      Area03_Messages.W.Msg[WngIndex + 0] := A0301_Ribaltatore.Warning.Ax.NotAutReady;
      Area03_Messages.W.Msg[WngIndex + 1] := A0301_Ribaltatore.Warning.Ax.Minus_CndMissing;
      Area03_Messages.W.Msg[WngIndex + 2] := A0301_Ribaltatore.Warning.Ax.Plus_CndMissing AND A0301_Ribaltatore.COut.Solleva_Rib.Work;
      Area03_Messages.W.Msg[WngIndex + 3] := A0301_Ribaltatore.Warning.Ax.S120_Warning;
      Area03_Messages.W.Msg[WngIndex + 4] := A0301_Ribaltatore.Warning.Ax.Ax_NotHomed;
      Area03_Messages.W.Msg[WngIndex + 5] := A0301_Ribaltatore.Warning.Ax.Ax_FlyingHome;
      Area03_Messages.W.Msg[WngIndex + 6] := A0301_Ribaltatore.Warning.Ax.Ax_SwLimitMinus;
      Area03_Messages.W.Msg[WngIndex + 7] := A0301_Ribaltatore.Warning.Ax.Ax_SwLimitPlus;
      Area03_Messages.W.Msg[WngIndex + 8] := A0301_Ribaltatore.Warning.OP_REST_MissingCnd;
      Area03_Messages.W.Msg[WngIndex + 9] := A0301_Ribaltatore.Warning.OP_WORK_MissingCnd;
      Area03_Messages.W.Msg[WngIndex + 10] := A0301_Ribaltatore.Warning.Solleva_Rib[1].NotAutReady;
      Area03_Messages.W.Msg[WngIndex + 11] := A0301_Ribaltatore.Warning.Solleva_Rib[1].PressureRunning_Timeout;
      Area03_Messages.W.Msg[WngIndex + 12] := A0301_Ribaltatore.Warning.Solleva_Rib[1].Rest_MissingExtEnable;
      Area03_Messages.W.Msg[WngIndex + 13] := A0301_Ribaltatore.Warning.Solleva_Rib[1].Work_MissingExtEnable;
      Area03_Messages.W.Msg[WngIndex + 14] := A0301_Ribaltatore.Warning.Solleva_Rib[1].Missing_Rest_Ls_ON[1];
      Area03_Messages.W.Msg[WngIndex + 15] := A0301_Ribaltatore.Warning.Solleva_Rib[1].Missing_Work_Ls_ON[1];
      Area03_Messages.W.Msg[WngIndex + 16] := A0301_Ribaltatore.Warning.Solleva_Rib[2].NotAutReady;
      Area03_Messages.W.Msg[WngIndex + 17] := A0301_Ribaltatore.Warning.Solleva_Rib[2].PressureRunning_Timeout;
      Area03_Messages.W.Msg[WngIndex + 18] := A0301_Ribaltatore.Warning.Solleva_Rib[2].Rest_MissingExtEnable;
      Area03_Messages.W.Msg[WngIndex + 19] := A0301_Ribaltatore.Warning.Solleva_Rib[2].Work_MissingExtEnable;
      Area03_Messages.W.Msg[WngIndex + 20] := A0301_Ribaltatore.Warning.Solleva_Rib[2].Missing_Rest_Ls_ON[1];
      Area03_Messages.W.Msg[WngIndex + 21] := A0301_Ribaltatore.Warning.Solleva_Rib[2].Missing_Work_Ls_ON[1];
      Area03_Messages.W.Msg[WngIndex + 22] := A0301_Ribaltatore.Warning.Solleva_Rib[3].NotAutReady;
      Area03_Messages.W.Msg[WngIndex + 23] := A0301_Ribaltatore.Warning.Solleva_Rib[3].PressureRunning_Timeout;
      Area03_Messages.W.Msg[WngIndex + 24] := A0301_Ribaltatore.Warning.Solleva_Rib[3].Rest_MissingExtEnable;
      Area03_Messages.W.Msg[WngIndex + 25] := A0301_Ribaltatore.Warning.Solleva_Rib[3].Work_MissingExtEnable;
      Area03_Messages.W.Msg[WngIndex + 26] := A0301_Ribaltatore.Warning.Solleva_Rib[3].Missing_Rest_Ls_ON[1];
      Area03_Messages.W.Msg[WngIndex + 27] := A0301_Ribaltatore.Warning.Solleva_Rib[3].Missing_Work_Ls_ON[1];
      Area03_Messages.W.Msg[WngIndex + 28] := A0301_Ribaltatore.Warning.Solleva_Rib[4].NotAutReady;
      Area03_Messages.W.Msg[WngIndex + 29] := A0301_Ribaltatore.Warning.Solleva_Rib[4].PressureRunning_Timeout;
      Area03_Messages.W.Msg[WngIndex + 30] := A0301_Ribaltatore.Warning.Solleva_Rib[4].Rest_MissingExtEnable;
      Area03_Messages.W.Msg[WngIndex + 31] := A0301_Ribaltatore.Warning.Solleva_Rib[4].Work_MissingExtEnable;
      Area03_Messages.W.Msg[WngIndex + 32] := A0301_Ribaltatore.Warning.Solleva_Rib[4].Missing_Rest_Ls_ON[1];
      Area03_Messages.W.Msg[WngIndex + 33] := A0301_Ribaltatore.Warning.Solleva_Rib[4].Missing_Work_Ls_ON[1];
      Area03_Messages.W.Msg[WngIndex + 34] := A0301_Ribaltatore.Warning.Solleva_Rib[5].NotAutReady;
      Area03_Messages.W.Msg[WngIndex + 35] := A0301_Ribaltatore.Warning.Solleva_Rib[5].PressureRunning_Timeout;
      Area03_Messages.W.Msg[WngIndex + 36] := A0301_Ribaltatore.Warning.Solleva_Rib[5].Rest_MissingExtEnable;
      Area03_Messages.W.Msg[WngIndex + 37] := A0301_Ribaltatore.Warning.Solleva_Rib[5].Work_MissingExtEnable;
      Area03_Messages.W.Msg[WngIndex + 38] := A0301_Ribaltatore.Warning.Solleva_Rib[5].Missing_Rest_Ls_ON[1];
      Area03_Messages.W.Msg[WngIndex + 39] := A0301_Ribaltatore.Warning.Solleva_Rib[5].Missing_Work_Ls_ON[1];
      Area03_Messages.W.Msg[WngIndex + 40] := A0301_Ribaltatore.Warning.Solleva_Rib[6].NotAutReady;
      Area03_Messages.W.Msg[WngIndex + 41] := A0301_Ribaltatore.Warning.Solleva_Rib[6].PressureRunning_Timeout;
      Area03_Messages.W.Msg[WngIndex + 42] := A0301_Ribaltatore.Warning.Solleva_Rib[6].Rest_MissingExtEnable;
      Area03_Messages.W.Msg[WngIndex + 43] := A0301_Ribaltatore.Warning.Solleva_Rib[6].Work_MissingExtEnable;
      Area03_Messages.W.Msg[WngIndex + 44] := A0301_Ribaltatore.Warning.Solleva_Rib[6].Missing_Rest_Ls_ON[1];
      Area03_Messages.W.Msg[WngIndex + 45] := A0301_Ribaltatore.Warning.Solleva_Rib[6].Missing_Work_Ls_ON[1];
      Area03_Messages.W.Msg[WngIndex + 46] := FALSE;
      Area03_Messages.W.Msg[WngIndex + 47] := FALSE;
      Area03_Messages.W.Msg[WngIndex + 48] := FALSE;
      Area03_Messages.W.Msg[WngIndex + 49] := FALSE;

      //Fermi P4
      //
      WngIndex := 280;

      Area03_Messages.W.Msg[WngIndex + 0] := A0301_Fermi_P4.Warning.Fermi[1].NotAutReady;
      Area03_Messages.W.Msg[WngIndex + 1] := A0301_Fermi_P4.Warning.Fermi[1].PressureRunning_Timeout;
      Area03_Messages.W.Msg[WngIndex + 2] := A0301_Fermi_P4.Warning.Fermi[1].Rest_MissingExtEnable;
      Area03_Messages.W.Msg[WngIndex + 3] := A0301_Fermi_P4.Warning.Fermi[1].Work_MissingExtEnable;
      Area03_Messages.W.Msg[WngIndex + 4] := A0301_Fermi_P4.Warning.Fermi[1].Missing_Rest_Ls_ON[1];
      Area03_Messages.W.Msg[WngIndex + 5] := A0301_Fermi_P4.Warning.Fermi[1].Missing_Work_Ls_ON[1];
      Area03_Messages.W.Msg[WngIndex + 6] := A0301_Fermi_P4.Warning.Fermi[2].NotAutReady;
      Area03_Messages.W.Msg[WngIndex + 7] := A0301_Fermi_P4.Warning.Fermi[2].PressureRunning_Timeout;
      Area03_Messages.W.Msg[WngIndex + 8] := A0301_Fermi_P4.Warning.Fermi[2].Rest_MissingExtEnable;
      Area03_Messages.W.Msg[WngIndex + 9] := A0301_Fermi_P4.Warning.Fermi[2].Work_MissingExtEnable;
      Area03_Messages.W.Msg[WngIndex + 10] := A0301_Fermi_P4.Warning.Fermi[2].Missing_Rest_Ls_ON[1];
      Area03_Messages.W.Msg[WngIndex + 11] := A0301_Fermi_P4.Warning.Fermi[2].Missing_Work_Ls_ON[1];
      Area03_Messages.W.Msg[WngIndex + 12] := A0301_Fermi_P4.Warning.Fermi[3].NotAutReady;
      Area03_Messages.W.Msg[WngIndex + 13] := A0301_Fermi_P4.Warning.Fermi[3].PressureRunning_Timeout;
      Area03_Messages.W.Msg[WngIndex + 14] := A0301_Fermi_P4.Warning.Fermi[3].Rest_MissingExtEnable;
      Area03_Messages.W.Msg[WngIndex + 15] := A0301_Fermi_P4.Warning.Fermi[3].Work_MissingExtEnable;
      Area03_Messages.W.Msg[WngIndex + 16] := A0301_Fermi_P4.Warning.Fermi[3].Missing_Rest_Ls_ON[1];
      Area03_Messages.W.Msg[WngIndex + 17] := A0301_Fermi_P4.Warning.Fermi[3].Missing_Work_Ls_ON[1];
      Area03_Messages.W.Msg[WngIndex + 18] := A0301_Fermi_P4.Warning.Fermi[4].NotAutReady;
      Area03_Messages.W.Msg[WngIndex + 19] := A0301_Fermi_P4.Warning.Fermi[4].PressureRunning_Timeout;
      Area03_Messages.W.Msg[WngIndex + 20] := A0301_Fermi_P4.Warning.Fermi[4].Rest_MissingExtEnable;
      Area03_Messages.W.Msg[WngIndex + 21] := A0301_Fermi_P4.Warning.Fermi[4].Work_MissingExtEnable;
      Area03_Messages.W.Msg[WngIndex + 22] := A0301_Fermi_P4.Warning.Fermi[4].Missing_Rest_Ls_ON[1];
      Area03_Messages.W.Msg[WngIndex + 23] := A0301_Fermi_P4.Warning.Fermi[4].Missing_Work_Ls_ON[1];
      Area03_Messages.W.Msg[WngIndex + 24] := A0301_Fermi_P4.Warning.Fermi[5].NotAutReady;
      Area03_Messages.W.Msg[WngIndex + 25] := A0301_Fermi_P4.Warning.Fermi[5].PressureRunning_Timeout;
      Area03_Messages.W.Msg[WngIndex + 26] := A0301_Fermi_P4.Warning.Fermi[5].Rest_MissingExtEnable;
      Area03_Messages.W.Msg[WngIndex + 27] := A0301_Fermi_P4.Warning.Fermi[5].Work_MissingExtEnable;
      Area03_Messages.W.Msg[WngIndex + 28] := A0301_Fermi_P4.Warning.Fermi[5].Missing_Rest_Ls_ON[1];
      Area03_Messages.W.Msg[WngIndex + 29] := A0301_Fermi_P4.Warning.Fermi[5].Missing_Work_Ls_ON[1];
      Area03_Messages.W.Msg[WngIndex + 30] := A0301_Fermi_P4.Warning.Fermi[6].NotAutReady;
      Area03_Messages.W.Msg[WngIndex + 31] := A0301_Fermi_P4.Warning.Fermi[6].PressureRunning_Timeout;
      Area03_Messages.W.Msg[WngIndex + 32] := A0301_Fermi_P4.Warning.Fermi[6].Rest_MissingExtEnable;
      Area03_Messages.W.Msg[WngIndex + 33] := A0301_Fermi_P4.Warning.Fermi[6].Work_MissingExtEnable;
      Area03_Messages.W.Msg[WngIndex + 34] := A0301_Fermi_P4.Warning.Fermi[6].Missing_Rest_Ls_ON[1];
      Area03_Messages.W.Msg[WngIndex + 35] := A0301_Fermi_P4.Warning.Fermi[6].Missing_Work_Ls_ON[1];
      Area03_Messages.W.Msg[WngIndex + 36] := FALSE;
      Area03_Messages.W.Msg[WngIndex + 37] := FALSE;
      Area03_Messages.W.Msg[WngIndex + 38] := A0301_Fermi_P4.Warning.OP_REST_MissingCnd;
      Area03_Messages.W.Msg[WngIndex + 39] := A0301_Fermi_P4.Warning.OP_WORK_MissingCnd;

      //Spintore Laterale
      //
      WngIndex := 330;

      Area03_Messages.W.Msg[WngIndex + 0] := A0301_Spintore_Lat.Warning.Vrt_1.NotAutReady;
      Area03_Messages.W.Msg[WngIndex + 1] := A0301_Spintore_Lat.Warning.Vrt_1.PressureRunning_Timeout;
      Area03_Messages.W.Msg[WngIndex + 2] := A0301_Spintore_Lat.Warning.Vrt_1.Rest_MissingExtEnable;
      Area03_Messages.W.Msg[WngIndex + 3] := A0301_Spintore_Lat.Warning.Vrt_1.Work_MissingExtEnable;
      Area03_Messages.W.Msg[WngIndex + 4] := A0301_Spintore_Lat.Warning.Vrt_1.Missing_Rest_Ls_ON[1];
      Area03_Messages.W.Msg[WngIndex + 5] := A0301_Spintore_Lat.Warning.Vrt_1.Missing_Work_Ls_ON[1];
      Area03_Messages.W.Msg[WngIndex + 6] := FALSE;
      Area03_Messages.W.Msg[WngIndex + 7] := A0301_Spintore_Lat.Warning.Orz_1.NotAutReady;;
      Area03_Messages.W.Msg[WngIndex + 8] := A0301_Spintore_Lat.Warning.Orz_1.PressureRunning_Timeout;
      Area03_Messages.W.Msg[WngIndex + 9] := A0301_Spintore_Lat.Warning.Orz_1.Rest_MissingExtEnable;
      Area03_Messages.W.Msg[WngIndex + 10] := A0301_Spintore_Lat.Warning.Orz_1.Work_MissingExtEnable;
      Area03_Messages.W.Msg[WngIndex + 11] := A0301_Spintore_Lat.Warning.Orz_1.Missing_Rest_Ls_ON[1];
      Area03_Messages.W.Msg[WngIndex + 12] := A0301_Spintore_Lat.Warning.Orz_1.Missing_Work_Ls_ON[1];
      Area03_Messages.W.Msg[WngIndex + 13] := FALSE;
      Area03_Messages.W.Msg[WngIndex + 14] := A0301_Spintore_Lat.Warning.Orz_1_AnalSens.SensorDisabled;
      Area03_Messages.W.Msg[WngIndex + 15] := A0301_Spintore_Lat.Warning.Orz_1_AnalSens.PresetNeed;;
      Area03_Messages.W.Msg[WngIndex + 16] := A0301_Spintore_Lat.Warning.Orz_1_AnalSens.SignalError;
      Area03_Messages.W.Msg[WngIndex + 17] := FALSE;
      Area03_Messages.W.Msg[WngIndex + 18] := A0301_Spintore_Lat.Warning.OP_REST_MissingCnd;
      Area03_Messages.W.Msg[WngIndex + 19] := A0301_Spintore_Lat.Warning.OP_WORK_MissingCnd;
      Area03_Messages.W.Msg[WngIndex + 20] := A0301_Spintore_Lat.Warning.Vrt_2.NotAutReady;;
      Area03_Messages.W.Msg[WngIndex + 21] := A0301_Spintore_Lat.Warning.Vrt_2.PressureRunning_Timeout;
      Area03_Messages.W.Msg[WngIndex + 22] := A0301_Spintore_Lat.Warning.Vrt_2.Rest_MissingExtEnable;
      Area03_Messages.W.Msg[WngIndex + 23] := A0301_Spintore_Lat.Warning.Vrt_2.Work_MissingExtEnable;
      Area03_Messages.W.Msg[WngIndex + 24] := A0301_Spintore_Lat.Warning.Vrt_2.Missing_Rest_Ls_ON[1];
      Area03_Messages.W.Msg[WngIndex + 25] := A0301_Spintore_Lat.Warning.Vrt_2.Missing_Work_Ls_ON[1];
      Area03_Messages.W.Msg[WngIndex + 26] := FALSE;
      Area03_Messages.W.Msg[WngIndex + 27] := A0301_Spintore_Lat.Warning.Orz_2.NotAutReady;
      Area03_Messages.W.Msg[WngIndex + 28] := A0301_Spintore_Lat.Warning.Orz_2.PressureRunning_Timeout;
      Area03_Messages.W.Msg[WngIndex + 29] := A0301_Spintore_Lat.Warning.Orz_2.Rest_MissingExtEnable;
      Area03_Messages.W.Msg[WngIndex + 30] := A0301_Spintore_Lat.Warning.Orz_2.Work_MissingExtEnable;
      Area03_Messages.W.Msg[WngIndex + 31] := A0301_Spintore_Lat.Warning.Orz_2.Missing_Rest_Ls_ON[1];
      Area03_Messages.W.Msg[WngIndex + 32] := A0301_Spintore_Lat.Warning.Orz_2.Missing_Work_Ls_ON[1];
      Area03_Messages.W.Msg[WngIndex + 33] := A0301_Spintore_Lat.Warning.Orz_2_AnalSens.SensorDisabled;
      Area03_Messages.W.Msg[WngIndex + 34] := A0301_Spintore_Lat.Warning.Orz_2_AnalSens.PresetNeed;
      Area03_Messages.W.Msg[WngIndex + 35] := A0301_Spintore_Lat.Warning.Orz_2_AnalSens.SignalError;
      Area03_Messages.W.Msg[WngIndex + 36] := A0301_Spintore_Lat.Warning.Finestre.SpinLat1_SpinLong_Stop;
      Area03_Messages.W.Msg[WngIndex + 37] := A0301_Spintore_Lat.Warning.Finestre.SpinLat2_SpinLong_Stop;


      //Spintore Longitudinale
      //
      WngIndex := 380;

      Area03_Messages.W.Msg[WngIndex + 0] := A0301_Spintore_Lat.Warning.Sollevatori[1].NotAutReady;
      Area03_Messages.W.Msg[WngIndex + 1] := A0301_Spintore_Lat.Warning.Sollevatori[1].PressureRunning_Timeout;
      Area03_Messages.W.Msg[WngIndex + 2] := A0301_Spintore_Lat.Warning.Sollevatori[1].Rest_MissingExtEnable;
      Area03_Messages.W.Msg[WngIndex + 3] := A0301_Spintore_Lat.Warning.Sollevatori[1].Work_MissingExtEnable;
      Area03_Messages.W.Msg[WngIndex + 4] := A0301_Spintore_Lat.Warning.Sollevatori[1].Missing_Rest_Ls_ON[1];
      Area03_Messages.W.Msg[WngIndex + 5] := A0301_Spintore_Lat.Warning.Sollevatori[1].Missing_Work_Ls_ON[1];
      Area03_Messages.W.Msg[WngIndex + 6] := FALSE;
      Area03_Messages.W.Msg[WngIndex + 7] := A0301_Spintore_Lat.Warning.Sollevatori[2].NotAutReady;;
      Area03_Messages.W.Msg[WngIndex + 8] := A0301_Spintore_Lat.Warning.Sollevatori[2].PressureRunning_Timeout;
      Area03_Messages.W.Msg[WngIndex + 9] := A0301_Spintore_Lat.Warning.Sollevatori[2].Rest_MissingExtEnable;
      Area03_Messages.W.Msg[WngIndex + 10] := A0301_Spintore_Lat.Warning.Sollevatori[2].Work_MissingExtEnable;
      Area03_Messages.W.Msg[WngIndex + 11] := A0301_Spintore_Lat.Warning.Sollevatori[2].Missing_Rest_Ls_ON[1];
      Area03_Messages.W.Msg[WngIndex + 12] := A0301_Spintore_Lat.Warning.Sollevatori[2].Missing_Work_Ls_ON[1];
      Area03_Messages.W.Msg[WngIndex + 13] := FALSE;
      Area03_Messages.W.Msg[WngIndex + 14] := A0301_Spintore_Lat.Warning.Sollevatori[3].NotAutReady;
      Area03_Messages.W.Msg[WngIndex + 15] := A0301_Spintore_Lat.Warning.Sollevatori[3].PressureRunning_Timeout;
      Area03_Messages.W.Msg[WngIndex + 16] := A0301_Spintore_Lat.Warning.Sollevatori[3].Rest_MissingExtEnable;
      Area03_Messages.W.Msg[WngIndex + 17] := A0301_Spintore_Lat.Warning.Sollevatori[3].Work_MissingExtEnable;
      Area03_Messages.W.Msg[WngIndex + 18] := A0301_Spintore_Lat.Warning.Sollevatori[3].Missing_Rest_Ls_ON[1];
      Area03_Messages.W.Msg[WngIndex + 19] := A0301_Spintore_Lat.Warning.Sollevatori[3].Missing_Work_Ls_ON[1];
      Area03_Messages.W.Msg[WngIndex + 20] := FALSE;
      Area03_Messages.W.Msg[WngIndex + 21] := A0301_Spintore_Lat.Warning.Sollevatori[4].NotAutReady;
      Area03_Messages.W.Msg[WngIndex + 22] := A0301_Spintore_Lat.Warning.Sollevatori[4].PressureRunning_Timeout;
      Area03_Messages.W.Msg[WngIndex + 23] := A0301_Spintore_Lat.Warning.Sollevatori[4].Rest_MissingExtEnable;
      Area03_Messages.W.Msg[WngIndex + 24] := A0301_Spintore_Lat.Warning.Sollevatori[4].Work_MissingExtEnable;
      Area03_Messages.W.Msg[WngIndex + 25] := A0301_Spintore_Lat.Warning.Sollevatori[4].Missing_Rest_Ls_ON[1];
      Area03_Messages.W.Msg[WngIndex + 26] := A0301_Spintore_Lat.Warning.Sollevatori[4].Missing_Work_Ls_ON[1];
      Area03_Messages.W.Msg[WngIndex + 27] := FALSE;
      Area03_Messages.W.Msg[WngIndex + 28] := A0301_Spintore_Lat.Warning.Sollevatori[5].NotAutReady;
      Area03_Messages.W.Msg[WngIndex + 29] := A0301_Spintore_Lat.Warning.Sollevatori[5].PressureRunning_Timeout;
      Area03_Messages.W.Msg[WngIndex + 30] := A0301_Spintore_Lat.Warning.Sollevatori[5].Rest_MissingExtEnable;
      Area03_Messages.W.Msg[WngIndex + 31] := A0301_Spintore_Lat.Warning.Sollevatori[5].Work_MissingExtEnable;
      Area03_Messages.W.Msg[WngIndex + 32] := A0301_Spintore_Lat.Warning.Sollevatori[5].Missing_Rest_Ls_ON[1];
      Area03_Messages.W.Msg[WngIndex + 33] := A0301_Spintore_Lat.Warning.Sollevatori[5].Missing_Work_Ls_ON[1];
      Area03_Messages.W.Msg[WngIndex + 34] := FALSE;
      Area03_Messages.W.Msg[WngIndex + 35] := A0301_Spintore_Lat.Warning.Sollevatori[6].NotAutReady;
      Area03_Messages.W.Msg[WngIndex + 36] := A0301_Spintore_Lat.Warning.Sollevatori[6].PressureRunning_Timeout;
      Area03_Messages.W.Msg[WngIndex + 37] := A0301_Spintore_Lat.Warning.Sollevatori[6].Rest_MissingExtEnable;
      Area03_Messages.W.Msg[WngIndex + 38] := A0301_Spintore_Lat.Warning.Sollevatori[6].Work_MissingExtEnable;
      Area03_Messages.W.Msg[WngIndex + 39] := A0301_Spintore_Lat.Warning.Sollevatori[6].Missing_Rest_Ls_ON[1];
      Area03_Messages.W.Msg[WngIndex + 40] := A0301_Spintore_Lat.Warning.Sollevatori[6].Missing_Work_Ls_ON[1];
      Area03_Messages.W.Msg[WngIndex + 41] := FALSE;
      Area03_Messages.W.Msg[WngIndex + 42] := A0301_Spintore_Lat.Warning.Sollevatori[7].NotAutReady;
      Area03_Messages.W.Msg[WngIndex + 43] := A0301_Spintore_Lat.Warning.Sollevatori[7].PressureRunning_Timeout;
      Area03_Messages.W.Msg[WngIndex + 44] := A0301_Spintore_Lat.Warning.Sollevatori[7].Rest_MissingExtEnable;
      Area03_Messages.W.Msg[WngIndex + 45] := A0301_Spintore_Lat.Warning.Sollevatori[7].Work_MissingExtEnable;
      Area03_Messages.W.Msg[WngIndex + 46] := A0301_Spintore_Lat.Warning.Sollevatori[7].Missing_Rest_Ls_ON[1];
      Area03_Messages.W.Msg[WngIndex + 47] := A0301_Spintore_Lat.Warning.Sollevatori[7].Missing_Work_Ls_ON[1];
      Area03_Messages.W.Msg[WngIndex + 48] := FALSE;
      Area03_Messages.W.Msg[WngIndex + 49] := FALSE;



      //Manager stazioni pareggiamento
      //
      WngIndex := 430;

      Area03_Messages.W.Msg[WngIndex + 0] := A0302_Manager.Warning.CheckBancoAccumulo;
      Area03_Messages.W.Msg[WngIndex + 1] := FALSE;
      Area03_Messages.W.Msg[WngIndex + 2] := FALSE;
      Area03_Messages.W.Msg[WngIndex + 3] := FALSE;
      Area03_Messages.W.Msg[WngIndex + 4] := FALSE;
      Area03_Messages.W.Msg[WngIndex + 5] := FALSE;
      Area03_Messages.W.Msg[WngIndex + 6] := FALSE;
      Area03_Messages.W.Msg[WngIndex + 7] := FALSE;
      Area03_Messages.W.Msg[WngIndex + 8] := FALSE;
      Area03_Messages.W.Msg[WngIndex + 9] := FALSE;

      //HU CYTROPACK
      //
      WngIndex := 440;

      Area03_Messages.W.Msg[WngIndex + 0] := FALSE;
      Area03_Messages.W.Msg[WngIndex + 1] := FALSE;
      Area03_Messages.W.Msg[WngIndex + 2] := FALSE;
      Area03_Messages.W.Msg[WngIndex + 3] := FALSE;
      Area03_Messages.W.Msg[WngIndex + 4] := FALSE;
      Area03_Messages.W.Msg[WngIndex + 5] := FALSE;
      Area03_Messages.W.Msg[WngIndex + 6] := FALSE;
      Area03_Messages.W.Msg[WngIndex + 7] := FALSE;
      Area03_Messages.W.Msg[WngIndex + 8] := FALSE;
      Area03_Messages.W.Msg[WngIndex + 9] := FALSE;
      Area03_Messages.W.Msg[WngIndex + 10] := FALSE;
      Area03_Messages.W.Msg[WngIndex + 11] := FALSE;
      Area03_Messages.W.Msg[WngIndex + 12] := FALSE;
      Area03_Messages.W.Msg[WngIndex + 13] := FALSE;
      Area03_Messages.W.Msg[WngIndex + 14] := FALSE;
      Area03_Messages.W.Msg[WngIndex + 15] := FALSE;
      Area03_Messages.W.Msg[WngIndex + 16] := FALSE;
      Area03_Messages.W.Msg[WngIndex + 17] := FALSE;
      Area03_Messages.W.Msg[WngIndex + 18] := FALSE;
      Area03_Messages.W.Msg[WngIndex + 19] := FALSE;

      //Spintore
      //
      WngIndex := 470;

      Area03_Messages.W.Msg[WngIndex + 0] := A0302_Spintore.Warning.Ax.NotAutReady;
      Area03_Messages.W.Msg[WngIndex + 1] := A0302_Spintore.Warning.Ax.Minus_CndMissing;
      Area03_Messages.W.Msg[WngIndex + 2] := A0302_Spintore.Warning.Ax.Plus_CndMissing;
      Area03_Messages.W.Msg[WngIndex + 3] := A0302_Spintore.Warning.Ax.S120_Warning;
      Area03_Messages.W.Msg[WngIndex + 4] := A0302_Spintore.Warning.Ax.Ax_NotHomed;
      Area03_Messages.W.Msg[WngIndex + 5] := A0302_Spintore.Warning.Ax.Ax_FlyingHome;
      Area03_Messages.W.Msg[WngIndex + 6] := A0302_Spintore.Warning.Ax.Ax_SwLimitMinus;
      Area03_Messages.W.Msg[WngIndex + 7] := A0302_Spintore.Warning.Ax.Ax_SwLimitPlus;
      Area03_Messages.W.Msg[WngIndex + 8] := FALSE;
      Area03_Messages.W.Msg[WngIndex + 9] := FALSE;
      Area03_Messages.W.Msg[WngIndex + 10] := A0302_Spintore.Warning.Vrt.NotAutReady;
      Area03_Messages.W.Msg[WngIndex + 11] := A0302_Spintore.Warning.Vrt.PressureRunning_Timeout;
      Area03_Messages.W.Msg[WngIndex + 12] := A0302_Spintore.Warning.Vrt.Rest_MissingExtEnable;
      Area03_Messages.W.Msg[WngIndex + 13] := A0302_Spintore.Warning.Vrt.Work_MissingExtEnable;
      Area03_Messages.W.Msg[WngIndex + 14] := A0302_Spintore.Warning.Vrt.Missing_Rest_Ls_ON[1];
      Area03_Messages.W.Msg[WngIndex + 15] := A0302_Spintore.Warning.Vrt.Missing_Work_Ls_ON[1];
      Area03_Messages.W.Msg[WngIndex + 16] := FALSE;
      Area03_Messages.W.Msg[WngIndex + 17] := FALSE;
      Area03_Messages.W.Msg[WngIndex + 18] := A0302_Spintore.Warning.Orz.NotAutReady;
      Area03_Messages.W.Msg[WngIndex + 19] := A0302_Spintore.Warning.Orz.PressureRunning_Timeout;
      Area03_Messages.W.Msg[WngIndex + 20] := A0302_Spintore.Warning.Orz.Rest_MissingExtEnable;
      Area03_Messages.W.Msg[WngIndex + 21] := A0302_Spintore.Warning.Orz.Work_MissingExtEnable;
      Area03_Messages.W.Msg[WngIndex + 22] := A0302_Spintore.Warning.Orz.Missing_Rest_Ls_ON[1];
      Area03_Messages.W.Msg[WngIndex + 23] := A0302_Spintore.Warning.Orz.Missing_Work_Ls_ON[1];
      Area03_Messages.W.Msg[WngIndex + 24] := FALSE;
      Area03_Messages.W.Msg[WngIndex + 25] := FALSE;
      Area03_Messages.W.Msg[WngIndex + 26] := A0302_Spintore.Warning.Orz_AnalSens.SensorDisabled;
      Area03_Messages.W.Msg[WngIndex + 27] := A0302_Spintore.Warning.Orz_AnalSens.PresetNeed;
      Area03_Messages.W.Msg[WngIndex + 28] := A0302_Spintore.Warning.Orz_AnalSens.SignalError;
      Area03_Messages.W.Msg[WngIndex + 29] := FALSE;
      Area03_Messages.W.Msg[WngIndex + 30] := FALSE;
      Area03_Messages.W.Msg[WngIndex + 31] := A0302_Spintore.Warning.OP_REST_MissingCnd;
      Area03_Messages.W.Msg[WngIndex + 32] := A0302_Spintore.Warning.OP_WORK_MissingCnd;

      //Bordatrice
      //
      WngIndex := 510;

      Area03_Messages.W.Msg[WngIndex + 0] := A0302_Bordatrice.Warning.Ax.NotAutReady;
      Area03_Messages.W.Msg[WngIndex + 1] := A0302_Bordatrice.Warning.Ax.Minus_CndMissing;
      Area03_Messages.W.Msg[WngIndex + 2] := A0302_Bordatrice.Warning.Ax.Plus_CndMissing;
      Area03_Messages.W.Msg[WngIndex + 3] := A0302_Bordatrice.Warning.Ax.S120_Warning;
      Area03_Messages.W.Msg[WngIndex + 4] := A0302_Bordatrice.Warning.Ax.Ax_NotHomed;
      Area03_Messages.W.Msg[WngIndex + 5] := A0302_Bordatrice.Warning.Ax.Ax_FlyingHome;
      Area03_Messages.W.Msg[WngIndex + 6] := A0302_Bordatrice.Warning.Ax.Ax_SwLimitMinus;
      Area03_Messages.W.Msg[WngIndex + 7] := A0302_Bordatrice.Warning.Ax.Ax_SwLimitPlus;
      Area03_Messages.W.Msg[WngIndex + 8] := A0302_Bordatrice.Warning.OP_REST_MissingCnd;
      Area03_Messages.W.Msg[WngIndex + 9] := A0302_Bordatrice.Warning.OP_WORK_MissingCnd;
      Area03_Messages.W.Msg[WngIndex + 10] := FALSE;
      Area03_Messages.W.Msg[WngIndex + 11] := FALSE;
      Area03_Messages.W.Msg[WngIndex + 12] := FALSE;
      Area03_Messages.W.Msg[WngIndex + 13] := FALSE;
      Area03_Messages.W.Msg[WngIndex + 14] := FALSE;
      Area03_Messages.W.Msg[WngIndex + 15] := FALSE;
      Area03_Messages.W.Msg[WngIndex + 16] := FALSE;
      Area03_Messages.W.Msg[WngIndex + 17] := FALSE;
      Area03_Messages.W.Msg[WngIndex + 18] := FALSE;
      Area03_Messages.W.Msg[WngIndex + 19] := FALSE;
      Area03_Messages.W.Msg[WngIndex + 20] := FALSE;


      //Rulliera
      //
      WngIndex := 540;

      Area03_Messages.W.Msg[WngIndex + 0] := A0302_Rulliera.Warning.Rulliera[1].NotAutReady;
      Area03_Messages.W.Msg[WngIndex + 1] := A0302_Rulliera.Warning.Rulliera[1].MissingCnd_Bkw;
      Area03_Messages.W.Msg[WngIndex + 2] := A0302_Rulliera.Warning.Rulliera[1].MissingCnd_Fwd;
      Area03_Messages.W.Msg[WngIndex + 3] := A0302_Rulliera.Warning.Rulliera[1].Ax.Drive;
      Area03_Messages.W.Msg[WngIndex + 4] := A0302_Rulliera.Warning.Rulliera[2].NotAutReady;
      Area03_Messages.W.Msg[WngIndex + 5] := A0302_Rulliera.Warning.Rulliera[2].MissingCnd_Bkw;
      Area03_Messages.W.Msg[WngIndex + 6] := A0302_Rulliera.Warning.Rulliera[2].MissingCnd_Fwd;
      Area03_Messages.W.Msg[WngIndex + 7] := A0302_Rulliera.Warning.Rulliera[2].Ax.Drive;
      Area03_Messages.W.Msg[WngIndex + 8] := A0302_Rulliera.Warning.OP_REST_MissingCnd;
      Area03_Messages.W.Msg[WngIndex + 9] := A0302_Rulliera.Warning.OP_WORK_MissingCnd;
      Area03_Messages.W.Msg[WngIndex + 10] := FALSE;
      Area03_Messages.W.Msg[WngIndex + 11] := FALSE;
      Area03_Messages.W.Msg[WngIndex + 12] := FALSE;
      Area03_Messages.W.Msg[WngIndex + 13] := FALSE;
      Area03_Messages.W.Msg[WngIndex + 14] := FALSE;
      Area03_Messages.W.Msg[WngIndex + 15] := FALSE;
      Area03_Messages.W.Msg[WngIndex + 16] := FALSE;
      Area03_Messages.W.Msg[WngIndex + 17] := FALSE;
      Area03_Messages.W.Msg[WngIndex + 18] := FALSE;
      Area03_Messages.W.Msg[WngIndex + 19] := FALSE;


      //Centratori
      //
      WngIndex := 560;

      Area03_Messages.W.Msg[WngIndex + 0] := A0302_Centratori.Warning.Centratore[1].NotAutReady;
      Area03_Messages.W.Msg[WngIndex + 1] := A0302_Centratori.Warning.Centratore[1].PressureRunning_Timeout;
      Area03_Messages.W.Msg[WngIndex + 2] := A0302_Centratori.Warning.Centratore[1].Rest_MissingExtEnable;
      Area03_Messages.W.Msg[WngIndex + 3] := A0302_Centratori.Warning.Centratore[1].Work_MissingExtEnable;
      Area03_Messages.W.Msg[WngIndex + 4] := A0302_Centratori.Warning.Centratore[1].Missing_Rest_Ls_ON[1];
      Area03_Messages.W.Msg[WngIndex + 5] := A0302_Centratori.Warning.Centratore[1].Missing_Work_Ls_ON[1];
      Area03_Messages.W.Msg[WngIndex + 6] := FALSE;
      Area03_Messages.W.Msg[WngIndex + 7] := FALSE;
      Area03_Messages.W.Msg[WngIndex + 8] := A0302_Centratori.Warning.Centratore[2].NotAutReady;
      Area03_Messages.W.Msg[WngIndex + 9] := A0302_Centratori.Warning.Centratore[2].PressureRunning_Timeout;
      Area03_Messages.W.Msg[WngIndex + 10] := A0302_Centratori.Warning.Centratore[2].Rest_MissingExtEnable;
      Area03_Messages.W.Msg[WngIndex + 11] := A0302_Centratori.Warning.Centratore[2].Work_MissingExtEnable;
      Area03_Messages.W.Msg[WngIndex + 12] := A0302_Centratori.Warning.Centratore[2].Missing_Rest_Ls_ON[1];
      Area03_Messages.W.Msg[WngIndex + 13] := A0302_Centratori.Warning.Centratore[2].Missing_Work_Ls_ON[1];
      Area03_Messages.W.Msg[WngIndex + 14] := FALSE;
      Area03_Messages.W.Msg[WngIndex + 15] := FALSE;
      Area03_Messages.W.Msg[WngIndex + 16] := A0302_Centratori.Warning.Centratore[3].NotAutReady;
      Area03_Messages.W.Msg[WngIndex + 17] := A0302_Centratori.Warning.Centratore[3].PressureRunning_Timeout;
      Area03_Messages.W.Msg[WngIndex + 18] := A0302_Centratori.Warning.Centratore[3].Rest_MissingExtEnable;
      Area03_Messages.W.Msg[WngIndex + 19] := A0302_Centratori.Warning.Centratore[3].Work_MissingExtEnable;
      Area03_Messages.W.Msg[WngIndex + 20] := A0302_Centratori.Warning.Centratore[3].Missing_Rest_Ls_ON[1];
      Area03_Messages.W.Msg[WngIndex + 21] := A0302_Centratori.Warning.Centratore[3].Missing_Work_Ls_ON[1];
      Area03_Messages.W.Msg[WngIndex + 22] := FALSE;
      Area03_Messages.W.Msg[WngIndex + 23] := FALSE;
      Area03_Messages.W.Msg[WngIndex + 24] := A0302_Centratori.Warning.Sollevamento[1].NotAutReady;
      Area03_Messages.W.Msg[WngIndex + 25] := A0302_Centratori.Warning.Sollevamento[1].PressureRunning_Timeout;
      Area03_Messages.W.Msg[WngIndex + 26] := A0302_Centratori.Warning.Sollevamento[1].Rest_MissingExtEnable;
      Area03_Messages.W.Msg[WngIndex + 27] := A0302_Centratori.Warning.Sollevamento[1].Work_MissingExtEnable;
      Area03_Messages.W.Msg[WngIndex + 28] := A0302_Centratori.Warning.Sollevamento[1].Missing_Rest_Ls_ON[1];
      Area03_Messages.W.Msg[WngIndex + 29] := A0302_Centratori.Warning.Sollevamento[1].Missing_Work_Ls_ON[1];
      Area03_Messages.W.Msg[WngIndex + 30] := FALSE;
      Area03_Messages.W.Msg[WngIndex + 31] := FALSE;
      Area03_Messages.W.Msg[WngIndex + 32] := A0302_Centratori.Warning.Sollevamento[2].NotAutReady;
      Area03_Messages.W.Msg[WngIndex + 33] := A0302_Centratori.Warning.Sollevamento[2].PressureRunning_Timeout;
      Area03_Messages.W.Msg[WngIndex + 34] := A0302_Centratori.Warning.Sollevamento[2].Rest_MissingExtEnable;
      Area03_Messages.W.Msg[WngIndex + 35] := A0302_Centratori.Warning.Sollevamento[2].Work_MissingExtEnable;
      Area03_Messages.W.Msg[WngIndex + 36] := A0302_Centratori.Warning.Sollevamento[2].Missing_Rest_Ls_ON[1];
      Area03_Messages.W.Msg[WngIndex + 37] := A0302_Centratori.Warning.Sollevamento[2].Missing_Work_Ls_ON[1];
      Area03_Messages.W.Msg[WngIndex + 38] := FALSE;
      Area03_Messages.W.Msg[WngIndex + 39] := FALSE;
      Area03_Messages.W.Msg[WngIndex + 40] := A0302_Centratori.Warning.Sollevamento[3].NotAutReady;
      Area03_Messages.W.Msg[WngIndex + 41] := A0302_Centratori.Warning.Sollevamento[3].PressureRunning_Timeout;
      Area03_Messages.W.Msg[WngIndex + 42] := A0302_Centratori.Warning.Sollevamento[3].Rest_MissingExtEnable;
      Area03_Messages.W.Msg[WngIndex + 43] := A0302_Centratori.Warning.Sollevamento[3].Work_MissingExtEnable;
      Area03_Messages.W.Msg[WngIndex + 44] := A0302_Centratori.Warning.Sollevamento[3].Missing_Rest_Ls_ON[1];
      Area03_Messages.W.Msg[WngIndex + 45] := A0302_Centratori.Warning.Sollevamento[3].Missing_Work_Ls_ON[1];
      Area03_Messages.W.Msg[WngIndex + 46] := FALSE;
      Area03_Messages.W.Msg[WngIndex + 47] := FALSE;
      Area03_Messages.W.Msg[WngIndex + 48] := A0302_Centratori.Warning.OP_REST_Centr_MissingCnd;
      Area03_Messages.W.Msg[WngIndex + 49] := A0302_Centratori.Warning.OP_WORK_Centr_MissingCnd;

      //Pareggiatore Coda
      //
      WngIndex := 610;

      Area03_Messages.W.Msg[WngIndex + 0] := A0302_PareggiatoreCoda.Warning.Ax.NotAutReady;
      Area03_Messages.W.Msg[WngIndex + 1] := A0302_PareggiatoreCoda.Warning.Ax.MissingCnd_Minus;
      Area03_Messages.W.Msg[WngIndex + 2] := A0302_PareggiatoreCoda.Warning.Ax.MissingCnd_Plus;
      Area03_Messages.W.Msg[WngIndex + 3] := A0302_PareggiatoreCoda.Warning.Ax.Ax_NotHomed;
      Area03_Messages.W.Msg[WngIndex + 4] := A0302_PareggiatoreCoda.Warning.Ax.Ax.SwLimitMinus;
      Area03_Messages.W.Msg[WngIndex + 5] := A0302_PareggiatoreCoda.Warning.Ax.Ax.SwLimitPlus;
      Area03_Messages.W.Msg[WngIndex + 6] := A0302_PareggiatoreCoda.Warning.Ax.S120.Drive;
      Area03_Messages.W.Msg[WngIndex + 7] := FALSE;
      Area03_Messages.W.Msg[WngIndex + 8] := FALSE;
      Area03_Messages.W.Msg[WngIndex + 9] := FALSE;
      Area03_Messages.W.Msg[WngIndex + 10] := A0302_PareggiatoreCoda.Warning.Bloccaggio.NotAutReady;
      Area03_Messages.W.Msg[WngIndex + 11] := A0302_PareggiatoreCoda.Warning.Bloccaggio.PressureRunning_Timeout;
      Area03_Messages.W.Msg[WngIndex + 12] := A0302_PareggiatoreCoda.Warning.Bloccaggio.Rest_MissingExtEnable;
      Area03_Messages.W.Msg[WngIndex + 13] := A0302_PareggiatoreCoda.Warning.Bloccaggio.Work_MissingExtEnable;
      Area03_Messages.W.Msg[WngIndex + 14] := A0302_PareggiatoreCoda.Warning.Bloccaggio.Missing_Rest_Ls_ON[1];
      Area03_Messages.W.Msg[WngIndex + 15] := A0302_PareggiatoreCoda.Warning.Bloccaggio.Missing_Work_Ls_ON[1];
      Area03_Messages.W.Msg[WngIndex + 16] := FALSE;
      Area03_Messages.W.Msg[WngIndex + 17] := FALSE;
      Area03_Messages.W.Msg[WngIndex + 18] := A0302_PareggiatoreCoda.Warning.BattutaVerticale.NotAutReady;
      Area03_Messages.W.Msg[WngIndex + 19] := A0302_PareggiatoreCoda.Warning.BattutaVerticale.PressureRunning_Timeout;
      Area03_Messages.W.Msg[WngIndex + 20] := A0302_PareggiatoreCoda.Warning.BattutaVerticale.Rest_MissingExtEnable;
      Area03_Messages.W.Msg[WngIndex + 21] := A0302_PareggiatoreCoda.Warning.BattutaVerticale.Work_MissingExtEnable;
      Area03_Messages.W.Msg[WngIndex + 22] := A0302_PareggiatoreCoda.Warning.BattutaVerticale.Missing_Rest_Ls_ON[1];
      Area03_Messages.W.Msg[WngIndex + 23] := A0302_PareggiatoreCoda.Warning.BattutaVerticale.Missing_Work_Ls_ON[1];
      Area03_Messages.W.Msg[WngIndex + 24] := FALSE;
      Area03_Messages.W.Msg[WngIndex + 25] := FALSE;
      Area03_Messages.W.Msg[WngIndex + 26] := A0302_PareggiatoreCoda.Warning.PareggiatoreLongitudinale.NotAutReady;
      Area03_Messages.W.Msg[WngIndex + 27] := A0302_PareggiatoreCoda.Warning.PareggiatoreLongitudinale.PressureRunning_Timeout;
      Area03_Messages.W.Msg[WngIndex + 28] := A0302_PareggiatoreCoda.Warning.PareggiatoreLongitudinale.Rest_MissingExtEnable;
      Area03_Messages.W.Msg[WngIndex + 29] := A0302_PareggiatoreCoda.Warning.PareggiatoreLongitudinale.Work_MissingExtEnable;
      Area03_Messages.W.Msg[WngIndex + 30] := A0302_PareggiatoreCoda.Warning.PareggiatoreLongitudinale.Missing_Rest_Ls_ON[1];
      Area03_Messages.W.Msg[WngIndex + 31] := A0302_PareggiatoreCoda.Warning.PareggiatoreLongitudinale.Missing_Work_Ls_ON[1];
      Area03_Messages.W.Msg[WngIndex + 32] := FALSE;
      Area03_Messages.W.Msg[WngIndex + 33] := FALSE;
      Area03_Messages.W.Msg[WngIndex + 34] := A0302_PareggiatoreCoda.Warning.PosPareggiatoreLong.SensorDisabled;
      Area03_Messages.W.Msg[WngIndex + 35] := A0302_PareggiatoreCoda.Warning.PosPareggiatoreLong.PresetNeed;
      Area03_Messages.W.Msg[WngIndex + 36] := A0302_PareggiatoreCoda.Warning.PosPareggiatoreLong.SignalError;
      Area03_Messages.W.Msg[WngIndex + 37] := FALSE;
      Area03_Messages.W.Msg[WngIndex + 38] := A0302_PareggiatoreCoda.Warning.SW_Limit_AntiCollision;
      Area03_Messages.W.Msg[WngIndex + 39] := A0302_PareggiatoreCoda.Warning.MissingCnd.OP_REST_Bloccaggio;
      Area03_Messages.W.Msg[WngIndex + 40] := A0302_PareggiatoreCoda.Warning.MissingCnd.OP_WORK_Bloccaggio;
      Area03_Messages.W.Msg[WngIndex + 41] := A0302_PareggiatoreCoda.Warning.MissingCnd.OP_REST_BattutaVrt;
      Area03_Messages.W.Msg[WngIndex + 42] := A0302_PareggiatoreCoda.Warning.MissingCnd.OP_WORK_BattutaVrt;
      Area03_Messages.W.Msg[WngIndex + 43] := A0302_PareggiatoreCoda.Warning.MissingCnd.OP_REST_PareggLong;
      Area03_Messages.W.Msg[WngIndex + 44] := A0302_PareggiatoreCoda.Warning.MissingCnd.OP_WORK_PareggLong;


      //Pareggiatore Testa
      //
      WngIndex := 660;

      Area03_Messages.W.Msg[WngIndex + 0] := A0302_PareggiatoreTesta.Warning.Ax.NotAutReady;
      Area03_Messages.W.Msg[WngIndex + 1] := A0302_PareggiatoreTesta.Warning.Ax.MissingCnd_Minus;
      Area03_Messages.W.Msg[WngIndex + 2] := A0302_PareggiatoreTesta.Warning.Ax.MissingCnd_Plus;
      Area03_Messages.W.Msg[WngIndex + 3] := A0302_PareggiatoreTesta.Warning.Ax.Ax_NotHomed;
      Area03_Messages.W.Msg[WngIndex + 4] := A0302_PareggiatoreTesta.Warning.Ax.Ax.SwLimitMinus;
      Area03_Messages.W.Msg[WngIndex + 5] := A0302_PareggiatoreTesta.Warning.Ax.Ax.SwLimitPlus;
      Area03_Messages.W.Msg[WngIndex + 6] := A0302_PareggiatoreTesta.Warning.Ax.S120.Drive;
      Area03_Messages.W.Msg[WngIndex + 7] := FALSE;
      Area03_Messages.W.Msg[WngIndex + 8] := FALSE;
      Area03_Messages.W.Msg[WngIndex + 9] := FALSE;
      Area03_Messages.W.Msg[WngIndex + 10] := A0302_PareggiatoreTesta.Warning.Bloccaggio.NotAutReady;
      Area03_Messages.W.Msg[WngIndex + 11] := A0302_PareggiatoreTesta.Warning.Bloccaggio.PressureRunning_Timeout;
      Area03_Messages.W.Msg[WngIndex + 12] := A0302_PareggiatoreTesta.Warning.Bloccaggio.Rest_MissingExtEnable;
      Area03_Messages.W.Msg[WngIndex + 13] := A0302_PareggiatoreTesta.Warning.Bloccaggio.Work_MissingExtEnable;
      Area03_Messages.W.Msg[WngIndex + 14] := A0302_PareggiatoreTesta.Warning.Bloccaggio.Missing_Rest_Ls_ON[1];
      Area03_Messages.W.Msg[WngIndex + 15] := A0302_PareggiatoreTesta.Warning.Bloccaggio.Missing_Rest_Ls_ON[2];
      Area03_Messages.W.Msg[WngIndex + 16] := A0302_PareggiatoreTesta.Warning.Bloccaggio.Missing_Work_Ls_ON[1];
      Area03_Messages.W.Msg[WngIndex + 17] := A0302_PareggiatoreTesta.Warning.Bloccaggio.Missing_Work_Ls_ON[2];
      Area03_Messages.W.Msg[WngIndex + 18] := A0302_PareggiatoreTesta.Warning.Sollevamento.NotAutReady;
      Area03_Messages.W.Msg[WngIndex + 19] := A0302_PareggiatoreTesta.Warning.Sollevamento.PressureRunning_Timeout;
      Area03_Messages.W.Msg[WngIndex + 20] := A0302_PareggiatoreTesta.Warning.Sollevamento.Rest_MissingExtEnable;
      Area03_Messages.W.Msg[WngIndex + 21] := A0302_PareggiatoreTesta.Warning.Sollevamento.Work_MissingExtEnable;
      Area03_Messages.W.Msg[WngIndex + 22] := A0302_PareggiatoreTesta.Warning.Sollevamento.Missing_Rest_Ls_ON[1];
      Area03_Messages.W.Msg[WngIndex + 23] := A0302_PareggiatoreTesta.Warning.Sollevamento.Missing_Work_Ls_ON[1];
      Area03_Messages.W.Msg[WngIndex + 24] := FALSE;
      Area03_Messages.W.Msg[WngIndex + 25] := FALSE;
      Area03_Messages.W.Msg[WngIndex + 26] := A0302_PareggiatoreTesta.Warning.Centraggio.NotAutReady;
      Area03_Messages.W.Msg[WngIndex + 27] := A0302_PareggiatoreTesta.Warning.Centraggio.PressureRunning_Timeout;
      Area03_Messages.W.Msg[WngIndex + 28] := A0302_PareggiatoreTesta.Warning.Centraggio.Rest_MissingExtEnable;
      Area03_Messages.W.Msg[WngIndex + 29] := A0302_PareggiatoreTesta.Warning.Centraggio.Work_MissingExtEnable;
      Area03_Messages.W.Msg[WngIndex + 30] := A0302_PareggiatoreTesta.Warning.Centraggio.Missing_Rest_Ls_ON[1];
      Area03_Messages.W.Msg[WngIndex + 31] := A0302_PareggiatoreTesta.Warning.Centraggio.Missing_Work_Ls_ON[1];
      Area03_Messages.W.Msg[WngIndex + 32] := FALSE;
      Area03_Messages.W.Msg[WngIndex + 33] := A0302_PareggiatoreTesta.Warning.SW_Limit_AntiCollision;
      Area03_Messages.W.Msg[WngIndex + 34] := A0302_PareggiatoreTesta.Warning.MissingCnd.OP_REST_Bloccaggio;
      Area03_Messages.W.Msg[WngIndex + 35] := A0302_PareggiatoreTesta.Warning.MissingCnd.OP_WORK_Bloccaggio;
      Area03_Messages.W.Msg[WngIndex + 36] := A0302_PareggiatoreTesta.Warning.MissingCnd.OP_REST_Centraggio;
      Area03_Messages.W.Msg[WngIndex + 37] := A0302_PareggiatoreTesta.Warning.MissingCnd.OP_WORK_Centraggio;
      Area03_Messages.W.Msg[WngIndex + 38] := A0302_PareggiatoreTesta.Warning.MissingCnd.OP_REST_Sollevamento;
      Area03_Messages.W.Msg[WngIndex + 39] := A0302_PareggiatoreTesta.Warning.MissingCnd.OP_WORK_Sollevamento;

      //Manipolatore
      //
      WngIndex := 700;

      Area03_Messages.W.Msg[WngIndex + 0] := A0302_Manipolatore.Warning.Testa.Ax.NotAutReady;
      Area03_Messages.W.Msg[WngIndex + 1] := A0302_Manipolatore.Warning.Testa.Ax.Minus_CndMissing;
      Area03_Messages.W.Msg[WngIndex + 2] := A0302_Manipolatore.Warning.Testa.Ax.Plus_CndMissing;
      Area03_Messages.W.Msg[WngIndex + 3] := A0302_Manipolatore.Warning.Testa.Ax.S120_Warning;
      Area03_Messages.W.Msg[WngIndex + 4] := A0302_Manipolatore.Warning.Testa.Ax.Ax_NotHomed;
      Area03_Messages.W.Msg[WngIndex + 5] := A0302_Manipolatore.Warning.Testa.Ax.Ax_FlyingHome;
      Area03_Messages.W.Msg[WngIndex + 6] := A0302_Manipolatore.Warning.Testa.Ax.Ax_SwLimitMinus;
      Area03_Messages.W.Msg[WngIndex + 7] := A0302_Manipolatore.Warning.Testa.Ax.Ax_SwLimitPlus;
      Area03_Messages.W.Msg[WngIndex + 8] := FALSE;
      Area03_Messages.W.Msg[WngIndex + 9] := FALSE;
      Area03_Messages.W.Msg[WngIndex + 10] := A0302_Manipolatore.Warning.Testa.Sollevatore.NotAutReady;
      Area03_Messages.W.Msg[WngIndex + 11] := A0302_Manipolatore.Warning.Testa.Sollevatore.PressureRunning_Timeout;
      Area03_Messages.W.Msg[WngIndex + 12] := A0302_Manipolatore.Warning.Testa.Sollevatore.Rest_MissingExtEnable;
      Area03_Messages.W.Msg[WngIndex + 13] := A0302_Manipolatore.Warning.Testa.Sollevatore.Work_MissingExtEnable;
      Area03_Messages.W.Msg[WngIndex + 14] := A0302_Manipolatore.Warning.Testa.Sollevatore.Missing_Rest_Ls_ON[1];
      Area03_Messages.W.Msg[WngIndex + 15] := A0302_Manipolatore.Warning.Testa.Sollevatore.Missing_Work_Ls_ON[1];
      Area03_Messages.W.Msg[WngIndex + 16] := FALSE;
      Area03_Messages.W.Msg[WngIndex + 17] := FALSE;
      Area03_Messages.W.Msg[WngIndex + 18] := A0302_Manipolatore.Warning.Testa.Magnete.NotAutReady;
      Area03_Messages.W.Msg[WngIndex + 19] := A0302_Manipolatore.Warning.Testa.Magnete.PressureRunning_Timeout;
      Area03_Messages.W.Msg[WngIndex + 20] := A0302_Manipolatore.Warning.Testa.Magnete.Rest_MissingExtEnable;
      Area03_Messages.W.Msg[WngIndex + 21] := A0302_Manipolatore.Warning.Testa.Magnete.Work_MissingExtEnable;
      Area03_Messages.W.Msg[WngIndex + 22] := A0302_Manipolatore.Warning.Testa.Magnete.Missing_Rest_Ls_ON[1];
      Area03_Messages.W.Msg[WngIndex + 23] := A0302_Manipolatore.Warning.Testa.Magnete.Missing_Work_Ls_ON[1];
      Area03_Messages.W.Msg[WngIndex + 24] := FALSE;
      Area03_Messages.W.Msg[WngIndex + 25] := FALSE;
      Area03_Messages.W.Msg[WngIndex + 26] := A0302_Manipolatore.Warning.Coda.Ax.NotAutReady;
      Area03_Messages.W.Msg[WngIndex + 27] := A0302_Manipolatore.Warning.Coda.Ax.Minus_CndMissing;
      Area03_Messages.W.Msg[WngIndex + 28] := A0302_Manipolatore.Warning.Coda.Ax.Plus_CndMissing;
      Area03_Messages.W.Msg[WngIndex + 29] := A0302_Manipolatore.Warning.Coda.Ax.S120_Warning;
      Area03_Messages.W.Msg[WngIndex + 30] := A0302_Manipolatore.Warning.Coda.Ax.Ax_NotHomed;
      Area03_Messages.W.Msg[WngIndex + 31] := A0302_Manipolatore.Warning.Coda.Ax.Ax_FlyingHome;
      Area03_Messages.W.Msg[WngIndex + 32] := A0302_Manipolatore.Warning.Coda.Ax.Ax_SwLimitMinus;
      Area03_Messages.W.Msg[WngIndex + 33] := A0302_Manipolatore.Warning.Coda.Ax.Ax_SwLimitPlus;
      Area03_Messages.W.Msg[WngIndex + 34] := FALSE;
      Area03_Messages.W.Msg[WngIndex + 35] := FALSE;
      Area03_Messages.W.Msg[WngIndex + 36] := A0302_Manipolatore.Warning.Coda.Sollevatore.NotAutReady;
      Area03_Messages.W.Msg[WngIndex + 37] := A0302_Manipolatore.Warning.Coda.Sollevatore.PressureRunning_Timeout;
      Area03_Messages.W.Msg[WngIndex + 38] := A0302_Manipolatore.Warning.Coda.Sollevatore.Rest_MissingExtEnable;
      Area03_Messages.W.Msg[WngIndex + 39] := A0302_Manipolatore.Warning.Coda.Sollevatore.Work_MissingExtEnable;
      Area03_Messages.W.Msg[WngIndex + 40] := A0302_Manipolatore.Warning.Coda.Sollevatore.Missing_Rest_Ls_ON[1];
      Area03_Messages.W.Msg[WngIndex + 41] := A0302_Manipolatore.Warning.Coda.Sollevatore.Missing_Work_Ls_ON[1];
      Area03_Messages.W.Msg[WngIndex + 42] := FALSE;
      Area03_Messages.W.Msg[WngIndex + 43] := FALSE;
      Area03_Messages.W.Msg[WngIndex + 44] := A0302_Manipolatore.Warning.Testa.Magnete.NotAutReady;
      Area03_Messages.W.Msg[WngIndex + 45] := A0302_Manipolatore.Warning.Testa.Magnete.PressureRunning_Timeout;
      Area03_Messages.W.Msg[WngIndex + 46] := A0302_Manipolatore.Warning.Testa.Magnete.Rest_MissingExtEnable;
      Area03_Messages.W.Msg[WngIndex + 47] := A0302_Manipolatore.Warning.Testa.Magnete.Work_MissingExtEnable;
      Area03_Messages.W.Msg[WngIndex + 48] := A0302_Manipolatore.Warning.Testa.Magnete.Missing_Rest_Ls_ON[1];
      Area03_Messages.W.Msg[WngIndex + 49] := A0302_Manipolatore.Warning.Testa.Magnete.Missing_Work_Ls_ON[1];
      Area03_Messages.W.Msg[WngIndex + 50] := A0302_Manipolatore.Warning.MissingCnd.OP_REST_Sollevamento;
      Area03_Messages.W.Msg[WngIndex + 51] := A0302_Manipolatore.Warning.MissingCnd.OP_WORK_Sollevamento;
      Area03_Messages.W.Msg[WngIndex + 52] := A0302_Manipolatore.Warning.MissingCnd.OP_REST_Magneti;
      Area03_Messages.W.Msg[WngIndex + 53] := A0302_Manipolatore.Warning.MissingCnd.OP_WORK_Magneti;

      //Regolazione Bordatrice
      //
      WngIndex := 760;

      Area03_Messages.W.Msg[WngIndex + 0] := A0302_Bordatrice_RegolazioneFormato.Warning.Ax_D[1].NotAutReady;
      Area03_Messages.W.Msg[WngIndex + 1] := A0302_Bordatrice_RegolazioneFormato.Warning.Ax_D[1].MissingCnd_Minus;
      Area03_Messages.W.Msg[WngIndex + 2] := A0302_Bordatrice_RegolazioneFormato.Warning.Ax_D[1].MissingCnd_Plus;
      Area03_Messages.W.Msg[WngIndex + 3] := A0302_Bordatrice_RegolazioneFormato.Warning.Ax_D[1].Ax_NotHomed;
      Area03_Messages.W.Msg[WngIndex + 4] := A0302_Bordatrice_RegolazioneFormato.Warning.Ax_D[1].Ax.SwLimitMinus;
      Area03_Messages.W.Msg[WngIndex + 5] := A0302_Bordatrice_RegolazioneFormato.Warning.Ax_D[1].Ax.SwLimitPlus;
      Area03_Messages.W.Msg[WngIndex + 6] := A0302_Bordatrice_RegolazioneFormato.Warning.Ax_D[1].S120.Drive;
      Area03_Messages.W.Msg[WngIndex + 7] := FALSE;
      Area03_Messages.W.Msg[WngIndex + 8] := A0302_Bordatrice_RegolazioneFormato.Warning.Ax_M[1].NotAutReady;
      Area03_Messages.W.Msg[WngIndex + 9] := A0302_Bordatrice_RegolazioneFormato.Warning.Ax_M[1].Minus_CndMissing;
      Area03_Messages.W.Msg[WngIndex + 10] := A0302_Bordatrice_RegolazioneFormato.Warning.Ax_M[1].Plus_CndMissing;
      Area03_Messages.W.Msg[WngIndex + 11] := A0302_Bordatrice_RegolazioneFormato.Warning.Ax_M[1].Ax_NotHomed;
      Area03_Messages.W.Msg[WngIndex + 12] := A0302_Bordatrice_RegolazioneFormato.Warning.Ax_M[1].Ax.SwLimitMinus;
      Area03_Messages.W.Msg[WngIndex + 13] := A0302_Bordatrice_RegolazioneFormato.Warning.Ax_M[1].Ax.SwLimitPlus;
      Area03_Messages.W.Msg[WngIndex + 14] := A0302_Bordatrice_RegolazioneFormato.Warning.Ax_M[2].NotAutReady;
      Area03_Messages.W.Msg[WngIndex + 15] := A0302_Bordatrice_RegolazioneFormato.Warning.Ax_M[2].Minus_CndMissing;
      Area03_Messages.W.Msg[WngIndex + 16] := A0302_Bordatrice_RegolazioneFormato.Warning.Ax_M[2].Plus_CndMissing;
      Area03_Messages.W.Msg[WngIndex + 17] := A0302_Bordatrice_RegolazioneFormato.Warning.Ax_M[2].Ax_NotHomed;
      Area03_Messages.W.Msg[WngIndex + 18] := A0302_Bordatrice_RegolazioneFormato.Warning.Ax_M[2].Ax.SwLimitMinus;
      Area03_Messages.W.Msg[WngIndex + 19] := A0302_Bordatrice_RegolazioneFormato.Warning.Ax_M[2].Ax.SwLimitPlus;
      Area03_Messages.W.Msg[WngIndex + 20] := A0302_Bordatrice_RegolazioneFormato.Warning.Ax_M[3].NotAutReady;
      Area03_Messages.W.Msg[WngIndex + 21] := A0302_Bordatrice_RegolazioneFormato.Warning.Ax_M[3].Minus_CndMissing;
      Area03_Messages.W.Msg[WngIndex + 22] := A0302_Bordatrice_RegolazioneFormato.Warning.Ax_M[3].Plus_CndMissing;
      Area03_Messages.W.Msg[WngIndex + 23] := A0302_Bordatrice_RegolazioneFormato.Warning.Ax_M[3].Ax_NotHomed;
      Area03_Messages.W.Msg[WngIndex + 24] := A0302_Bordatrice_RegolazioneFormato.Warning.Ax_M[3].Ax.SwLimitMinus;
      Area03_Messages.W.Msg[WngIndex + 25] := A0302_Bordatrice_RegolazioneFormato.Warning.Ax_M[3].Ax.SwLimitPlus;
      Area03_Messages.W.Msg[WngIndex + 26] := A0302_Bordatrice_RegolazioneFormato.Warning.Ax_M[4].NotAutReady;
      Area03_Messages.W.Msg[WngIndex + 27] := A0302_Bordatrice_RegolazioneFormato.Warning.Ax_M[4].Minus_CndMissing;
      Area03_Messages.W.Msg[WngIndex + 28] := A0302_Bordatrice_RegolazioneFormato.Warning.Ax_M[4].Plus_CndMissing;
      Area03_Messages.W.Msg[WngIndex + 29] := A0302_Bordatrice_RegolazioneFormato.Warning.Ax_M[4].Ax_NotHomed;
      Area03_Messages.W.Msg[WngIndex + 30] := A0302_Bordatrice_RegolazioneFormato.Warning.Ax_M[4].Ax.SwLimitMinus;
      Area03_Messages.W.Msg[WngIndex + 31] := A0302_Bordatrice_RegolazioneFormato.Warning.Ax_M[4].Ax.SwLimitPlus;
      Area03_Messages.W.Msg[WngIndex + 32] := A0302_Bordatrice_RegolazioneFormato.Warning.Ax_M[5].NotAutReady;
      Area03_Messages.W.Msg[WngIndex + 33] := A0302_Bordatrice_RegolazioneFormato.Warning.Ax_M[5].Minus_CndMissing;
      Area03_Messages.W.Msg[WngIndex + 34] := A0302_Bordatrice_RegolazioneFormato.Warning.Ax_M[5].Plus_CndMissing;
      Area03_Messages.W.Msg[WngIndex + 35] := A0302_Bordatrice_RegolazioneFormato.Warning.Ax_M[5].Ax_NotHomed;
      Area03_Messages.W.Msg[WngIndex + 36] := A0302_Bordatrice_RegolazioneFormato.Warning.Ax_M[5].Ax.SwLimitMinus;
      Area03_Messages.W.Msg[WngIndex + 37] := A0302_Bordatrice_RegolazioneFormato.Warning.Ax_M[5].Ax.SwLimitPlus;
      Area03_Messages.W.Msg[WngIndex + 38] := A0302_Bordatrice_RegolazioneFormato.Warning.Ax_M[6].NotAutReady;
      Area03_Messages.W.Msg[WngIndex + 39] := A0302_Bordatrice_RegolazioneFormato.Warning.Ax_M[6].Minus_CndMissing;
      Area03_Messages.W.Msg[WngIndex + 40] := A0302_Bordatrice_RegolazioneFormato.Warning.Ax_M[6].Plus_CndMissing;
      Area03_Messages.W.Msg[WngIndex + 41] := A0302_Bordatrice_RegolazioneFormato.Warning.Ax_M[6].Ax_NotHomed;
      Area03_Messages.W.Msg[WngIndex + 42] := A0302_Bordatrice_RegolazioneFormato.Warning.Ax_M[6].Ax.SwLimitMinus;
      Area03_Messages.W.Msg[WngIndex + 43] := A0302_Bordatrice_RegolazioneFormato.Warning.Ax_M[6].Ax.SwLimitPlus;
      Area03_Messages.W.Msg[WngIndex + 44] := A0302_Bordatrice_RegolazioneFormato.Warning.Ax_M[7].NotAutReady;
      Area03_Messages.W.Msg[WngIndex + 45] := A0302_Bordatrice_RegolazioneFormato.Warning.Ax_M[7].Minus_CndMissing;
      Area03_Messages.W.Msg[WngIndex + 46] := A0302_Bordatrice_RegolazioneFormato.Warning.Ax_M[7].Plus_CndMissing;
      Area03_Messages.W.Msg[WngIndex + 47] := A0302_Bordatrice_RegolazioneFormato.Warning.Ax_M[7].Ax_NotHomed;
      Area03_Messages.W.Msg[WngIndex + 48] := A0302_Bordatrice_RegolazioneFormato.Warning.Ax_M[7].Ax.SwLimitMinus;
      Area03_Messages.W.Msg[WngIndex + 49] := A0302_Bordatrice_RegolazioneFormato.Warning.Ax_M[7].Ax.SwLimitPlus;
      Area03_Messages.W.Msg[WngIndex + 50] := A0302_Bordatrice_RegolazioneFormato.Warning.Ax_M[8].NotAutReady;
      Area03_Messages.W.Msg[WngIndex + 51] := A0302_Bordatrice_RegolazioneFormato.Warning.Ax_M[8].Minus_CndMissing;
      Area03_Messages.W.Msg[WngIndex + 52] := A0302_Bordatrice_RegolazioneFormato.Warning.Ax_M[8].Plus_CndMissing;
      Area03_Messages.W.Msg[WngIndex + 53] := A0302_Bordatrice_RegolazioneFormato.Warning.Ax_M[8].Ax_NotHomed;
      Area03_Messages.W.Msg[WngIndex + 54] := A0302_Bordatrice_RegolazioneFormato.Warning.Ax_M[8].Ax.SwLimitMinus;
      Area03_Messages.W.Msg[WngIndex + 55] := A0302_Bordatrice_RegolazioneFormato.Warning.Ax_M[8].Ax.SwLimitPlus;
      Area03_Messages.W.Msg[WngIndex + 56] := A0302_Bordatrice_RegolazioneFormato.Warning.Ax_M[9].NotAutReady;
      Area03_Messages.W.Msg[WngIndex + 57] := A0302_Bordatrice_RegolazioneFormato.Warning.Ax_M[9].Minus_CndMissing;
      Area03_Messages.W.Msg[WngIndex + 58] := A0302_Bordatrice_RegolazioneFormato.Warning.Ax_M[9].Plus_CndMissing;
      Area03_Messages.W.Msg[WngIndex + 59] := A0302_Bordatrice_RegolazioneFormato.Warning.Ax_M[9].Ax_NotHomed;
      Area03_Messages.W.Msg[WngIndex + 60] := A0302_Bordatrice_RegolazioneFormato.Warning.Ax_M[9].Ax.SwLimitMinus;
      Area03_Messages.W.Msg[WngIndex + 61] := A0302_Bordatrice_RegolazioneFormato.Warning.Ax_M[9].Ax.SwLimitPlus;
      Area03_Messages.W.Msg[WngIndex + 62] := FALSE;
      Area03_Messages.W.Msg[WngIndex + 63] := A0302_Bordatrice_RegolazioneFormato.Warning.Passaggio01_MaxDisallineamentoAXs;
      Area03_Messages.W.Msg[WngIndex + 64] := A0302_Bordatrice_RegolazioneFormato.Warning.Passaggio02_MaxDisallineamentoAXs;
      Area03_Messages.W.Msg[WngIndex + 65] := A0302_Bordatrice_RegolazioneFormato.Warning.Passaggio03_MaxDisallineamentoAXs;
      Area03_Messages.W.Msg[WngIndex + 66] := A0302_Bordatrice_RegolazioneFormato.Warning.Passaggio04_MaxDisallineamentoAXs;
      Area03_Messages.W.Msg[WngIndex + 67] := FALSE;
      Area03_Messages.W.Msg[WngIndex + 68] := FALSE;
      Area03_Messages.W.Msg[WngIndex + 69] := FALSE;


      // Finale 829


      //
      "Area03_Messages".W.Msg[#WngIndex + 0] := FALSE;
      "Area03_Messages".W.Msg[#WngIndex + 1] := FALSE;
      "Area03_Messages".W.Msg[#WngIndex + 2] := FALSE;
      "Area03_Messages".W.Msg[#WngIndex + 3] := FALSE;
      "Area03_Messages".W.Msg[#WngIndex + 4] := FALSE;
      "Area03_Messages".W.Msg[#WngIndex + 5] := FALSE;
      "Area03_Messages".W.Msg[#WngIndex + 6] := FALSE;
      "Area03_Messages".W.Msg[#WngIndex + 7] := FALSE;
      "Area03_Messages".W.Msg[#WngIndex + 8] := FALSE;
      "Area03_Messages".W.Msg[#WngIndex + 9] := FALSE;
      "Area03_Messages".W.Msg[#WngIndex + 10] := FALSE;
      "Area03_Messages".W.Msg[#WngIndex + 11] := FALSE;
      "Area03_Messages".W.Msg[#WngIndex + 12] := FALSE;
      "Area03_Messages".W.Msg[#WngIndex + 13] := FALSE;
      "Area03_Messages".W.Msg[#WngIndex + 14] := FALSE;
      "Area03_Messages".W.Msg[#WngIndex + 15] := FALSE;
      "Area03_Messages".W.Msg[#WngIndex + 16] := FALSE;
      "Area03_Messages".W.Msg[#WngIndex + 17] := FALSE;
      "Area03_Messages".W.Msg[#WngIndex + 18] := FALSE;
      "Area03_Messages".W.Msg[#WngIndex + 19] := FALSE;
      "Area03_Messages".W.Msg[#WngIndex + 20] := FALSE;
      "Area03_Messages".W.Msg[#WngIndex + 21] := FALSE;
      "Area03_Messages".W.Msg[#WngIndex + 22] := FALSE;
      "Area03_Messages".W.Msg[#WngIndex + 23] := FALSE;
      "Area03_Messages".W.Msg[#WngIndex + 24] := FALSE;
      "Area03_Messages".W.Msg[#WngIndex + 25] := FALSE;
      "Area03_Messages".W.Msg[#WngIndex + 26] := FALSE;
      "Area03_Messages".W.Msg[#WngIndex + 27] := FALSE;
      "Area03_Messages".W.Msg[#WngIndex + 28] := FALSE;
      "Area03_Messages".W.Msg[#WngIndex + 29] := FALSE;
      "Area03_Messages".W.Msg[#WngIndex + 30] := FALSE;
      "Area03_Messages".W.Msg[#WngIndex + 31] := FALSE;
      "Area03_Messages".W.Msg[#WngIndex + 32] := FALSE;
      "Area03_Messages".W.Msg[#WngIndex + 33] := FALSE;
      "Area03_Messages".W.Msg[#WngIndex + 34] := FALSE;
      "Area03_Messages".W.Msg[#WngIndex + 35] := FALSE;
      "Area03_Messages".W.Msg[#WngIndex + 36] := FALSE;
      "Area03_Messages".W.Msg[#WngIndex + 37] := FALSE;
      "Area03_Messages".W.Msg[#WngIndex + 38] := FALSE;
      "Area03_Messages".W.Msg[#WngIndex + 39] := FALSE;


   END_REGION

   REGION "Warnings manager"
      #Area03_Msg_Warnings(
         en := TRUE,
         Ack := Area03.DataIn.PbAckRst,
         Messages := Area03_Messages.W.Msg,
         MessagesHMI := Area03_Messages.W.Hmi,
         MessagesACK := Area03_Messages.W.Ack,
         MessageCount => A03_HMI.Area03.Status.WarningsNumber
      );

      #Area03_Msg_Warnings.Q;
   END_REGION

   REGION "MB lamp indicators"
      MB3_Lp_Abilitazione_Automatico_Area03 := Area03.DataOut.lampReady;
      MB3_Lp_Start_Ciclo_Area03 := Area03.DataOut.lampCycle;
      MB3_Lp_Reset_Anomalie := ((NOT ((NOT (Area03.DataOut.LampAlarmPresence) AND NOT (Area03.DataOut.LampWarningPresence))) AND Sys.Clock_1S) OR (NOT ((NOT (Area03.DataOut.LampAlarmPresence) AND NOT (Area03.DataOut.LampWarningPresence))) AND NOT (Area03_Msg_Alarms.NewMessage)));
      MB3_Lp_Avanti_Stazione_1_Area03 := MB3_Pb_Avanti_Stazione_1_Area03;
      MB3_Lp_Avanti_Stazione_2_Area03 := MB3_Pb_Avanti_Stazione_2_Area03;
   END_REGION

   REGION "Super User"
      A03_HMI.Area03.SuperUser.SgnMan := Area03.AreaInterface.Man;
      A03_HMI.Area03.SuperUser.SgnAut := Area03.AreaInterface.Aut;
      A03_HMI.Area03.SuperUser.SgnReset := A03_HMI.Area03.SuperUser.PbReset;
      A03_HMI.Area03.SuperUser.SgnStart := Area03.AreaInterface.Cycle;
      A03_HMI.Area03.SuperUser.SgnWngPresence := (A03_HMI.Area03.Status.WarningsNumber > 0);
      A03_HMI.Area03.SuperUser.SgnAlrPresence := (A03_HMI.Area03.Status.AlarmsNumber > 0);
      A03_HMI.Area03.SuperUser.SgnMessagePresence := false;
      A03_HMI.Area03.SuperUser.SgnStop := NOT ((NOT (Area03.AreaInterface.StopInPhase) AND NOT (Area03.AreaInterface.StopProgrammed)));
   END_REGION

   REGION "<<< MACHINES AREA 03 >>>"
      // Gen
      A03_HMI_CALL();



      // A0301
      // //
      A0301_Manager_CALL();

      A0301_Trasporto_CALL();

      A0301_Fermi_P1_CALL();

      A0301_Fermi_P2_CALL();

      A0301_Fermi_P3_CALL();

      A0301_Ribaltatore_CALL();

      A0301_Fermi_P4_CALL();

      A0301_Spintore_Lat_CALL();

      //A0302
      //
      A0302_Manager_CALL();

      A0302_HU_Cytropack_CALL();

      A0302_Spintore_CALL();

      A0302_Bordatrice_CALL();

      A0302_Bordatrice_RegolazioneFormato_OB1_CALL();

      A0302_Rulliera_CALL();

      A0302_Centratori_CALL();

      A0302_PareggiatoreCoda_CALL();

      A0302_PareggiatoreTesta_CALL();

      A0302_Manipolatore_CALL();



      A03_TrkManager_CALL();











   END_REGION

   REGION "AREA ITF"
      "Area03_ITF"(
         en := TRUE
      );

      "Area03_ITF"();
   END_REGION

   REGION "Entry enable Z21 (RIBALTAMENTO)"
      Areas_ITF.A03.Safety_EntryEnable.Z21 := ((A0301_Trasporto.MachineInterface.MotionsStandStill AND A0301_Ribaltatore.MachineInterface.MotionsStandStill) AND A0302_Spintore.MachineInterface.MotionsStandStill);
   END_REGION

   REGION "Entry enable Z23 (BORDATRICE)"
      Areas_ITF.A03.Safety_EntryEnable.Z23 := (A0302_Bordatrice.MachineInterface.MotionsStandStill AND A0302_Bordatrice_RegolazioneFormato.MachineInterface.MotionsStandStill);
   END_REGION

   REGION "Entry enable Z23 (PAREGGIAMENTO)"
      Areas_ITF.A03.Safety_EntryEnable.Z25 := (((A0302_Rulliera.MachineInterface.MotionsStandStill AND A0302_PareggiatoreTesta.MachineInterface.MotionsStandStill) AND A0302_PareggiatoreCoda.MachineInterface.MotionsStandStill) AND A0302_Manipolatore.MachineInterface.MotionsStandStill);
   END_REGION


END_FUNCTION
